(* IEC 61131-3 sources: ST-graph-rag-mcp/test/fixtures/indexer-test, 4 files *)

(* ---- FB_Base.st ---- *)
FUNCTION_BLOCK FB_Base
VAR_INPUT
  Enable : BOOL;
END_VAR
VAR_OUTPUT
  Status : INT;
END_VAR
VAR
  Internal : INT;
END_VAR
  Internal := 0;
END_FUNCTION_BLOCK

(* ---- FB_Extended.st ---- *)
FUNCTION_BLOCK FB_Extended EXTENDS FB_Base IMPLEMENTS I_Ctrl
VAR_INPUT
  SetPoint : REAL;
END_VAR
VAR_OUTPUT
  Output : REAL;
END_VAR
VAR
  Helper : FB_Helper;
END_VAR
  Helper();
END_FUNCTION_BLOCK

(* ---- FB_Helper.st ---- *)
FUNCTION_BLOCK FB_Helper
VAR_INPUT
  Data : INT;
END_VAR
VAR_OUTPUT
  Result : BOOL;
END_VAR
  Result := Data > 0;
END_FUNCTION_BLOCK

(* ---- PRG_Main.st ---- *)
PROGRAM PRG_Main
VAR
  Controller : FB_Extended;
  Base : FB_Base;
END_VAR
  Base(Enable := TRUE);
  Controller(SetPoint := 50.0);
END_PROGRAM
